(* CoDeSys 2.3.9.35 project: Controle de Nível com sensor analógico e IHM.pro *)
(* Author: Altus *)
(* Libraries: DU35x.lib 7.7.11 15:59:13, Navigation.lib 15.7.11 10:06:00, SysLibTargetVisu.lib 26.11.08 09:53:28, Standard.lib 26.11.08 09:46:20, Iecsfc.lib 26.11.08 09:46:14, SYSLIBCALLBACK.LIB 26.11.08 09:53:30 *)

(* PLC configuration (modules and I/O channels)
Comunicação [Comunica] node 0, in %IB0 out %QB0
  COM1 [COM1] node 0, in %IB0 out %QB0 {BaudRate = 115200; Paridade = Sem Paridade; StopBits = 1 Stop Bit; Modem = Sem RTS/CTS; Delay = 5}
    MToolIEC [Codesys] node 0, in %IB0 out %QB0
  COM2 [COM2] node 1, in %IB0 out %QB0 {BaudRate = 115200; Paridade = Sem Paridade; StopBits = 1 Stop Bit; Modem = Sem RTS/CTS; Delay = 5}
    Desabilitada [Desabilitado485] node 0, in %IB0 out %QB0
Entradas Digitais 0 [Entradas0] node 0, in %IW0 out %QB0
  I00 AT %IX0.0 [BitInput] I0.0
  I01 AT %IX0.1 [BitInput] I0.1
  I02 AT %IX0.2 [BitInput] I0.2
  I03 AT %IX0.3 [BitInput] I0.3
  I04 AT %IX0.4 [BitInput] I0.4
  I05 AT %IX0.5 [BitInput] I0.5
  I06 AT %IX0.6 [BitInput] I0.6
  I07 AT %IX0.7 [BitInput] I0.7
  I08 AT %IX0.8 [BitInput] I0.8
Entradas Digitais 1 [Entradas1] node 0, in %IW1 out %QB0
  I10 AT %IX1.0 [BitInput] I1.0
  I11 AT %IX1.1 [BitInput] I1.1
  I12 AT %IX1.2 [BitInput] I1.2
  I13 AT %IX1.3 [BitInput] I1.3
  I14 AT %IX1.4 [BitInput] I1.4
  I15 AT %IX1.5 [BitInput] I1.5
  I16 AT %IX1.6 [BitInput] I1.6
  I17 AT %IX1.7 [BitInput] I1.7
  I18 AT %IX1.8 [BitInput] I1.8
Entradas Digitais 2 [Entradas2] node 0, in %IW2 out %QB0
  I20 AT %IX2.0 [BitInput] I2.0
  I21 AT %IX2.1 [BitInput] I2.1
AI0 AT %IW4 [WordInput] AI0 {TipoAnalogica = Tensão 0-10V; FiltroAnalogica = Filtro 0 - AI=2ms  / AV=90ms; FundoEscala = 100}
AI1 AT %IW5 [WordInput] AI1 {TipoAnalogica = Channel Disable; FiltroAnalogica = Filter 0 - AI=2ms  / AV=90ms; FundoEscala = 0}
AI2 AT %IW6 [WordInput] AI2 {TipoAnalogica = Channel Disable; FiltroAnalogica = Filter 0 - AI=2ms  / AV=90ms; FundoEscala = 0}
AI3 AT %IW7 [WordInput] AI3 {TipoAnalogica = Channel Disable; FiltroAnalogica = Filter 0 - AI=2ms  / AV=90ms; FundoEscala = 0}
Entradas Rápidas [EntradasRapidas] node 1, in %IB16 out %QB0
  Bloco 0 [Bloco0] node 0, in %IB16 out %QB0
    Desabilitado [DesabilitadoBloco0] node 0, in %IB16 out %QB0
  Bloco 1 [Bloco1] node 1, in %IB16 out %QB0
    Desabilitado [DesabilitadoBloco1] node 0, in %IB16 out %QB0
  Entrada Configuravél Bloco 0 [EntradaConfiBloco0] node 2, in %IB16 out %QB0
    Contador 0 [EntradaConfContador0] node 0, in %IB16 out %QB0 {EntradaConfiguravelContador = Disable}
  Entrada Configuravél Bloco 1 [EntradaConfiBloco1] node 3, in %IB16 out %QB0
    Contador 2 [EntradaConfContador2] node 0, in %IB16 out %QB0 {EntradaConfiguravelContador = Disable}
Saídas [Saidas] node 1, in %IB13 out %QB0
  Saídas Digitais 0 [Saidas0] node 0, in %IW0 out %QW0
    Q00 AT %QX0.0 [BitOutput] Q0.0
    Q01 AT %QX0.1 [BitOutput] Q0.1
    Q02 AT %QX0.2 [BitOutput] Q0.2
    Q03 AT %QX0.3 [BitOutput] Q0.3
    Q04 AT %QX0.4 [BitOutput] Q0.4
    Q05 AT %QX0.5 [BitOutput] Q0.5
    Q06 AT %QX0.6 [BitOutput] Q0.6
    Q07 AT %QX0.7 [BitOutput] Q0.7
  Saídas Digitais 1 [Saidas1] node 0, in %IW0 out %QW1
    Q10 AT %QX1.0 [BitOutput] Q1.0
    Q11 AT %QX1.1 [BitOutput] Q1.1
    Q12 AT %QX1.2 [BitOutput] Q1.2
    Q13 AT %QX1.3 [BitOutput] Q1.3
    Q14 AT %QX1.4 [BitOutput] Q1.4
    Q15 AT %QX1.5 [BitOutput] Q1.5
    Q16 AT %QX1.6 [BitOutput] Q1.6
    Q17 AT %QX1.7 [BitOutput] Q1.7
  Saídas Analógicas [SaidaAnalogica] node 0, in %IW0 out %QW3
    AO0 AT %QW3 [WordOutput] AO0 {TipoAnalogica = Channel Disable; FundoEscala = 0}
    AO1 AT %QW4 [WordOutput] AO1 {TipoAnalogica = Channel Disable; FundoEscala = 0}
  Saídas Rápidas [SaidasRapidas] node 1, in %IB0 out %QB10
    Saída Rápida 0 Desabilitada [DesabilitadoF0] node 0, in %IB0 out %QB10
    Saída Rápida 1 Desabilitada [DesabilitadoF1] node 1, in %IB0 out %QB10
  Saídas Comum de Contador [SaidasContador] node 2, in %IB0 out %QB10
    Saída do Bloco 0 Desabilitada [DesabilitadoSaidaBloco0] node 0, in %IB0 out %QB10
    Saída do Bloco 1 Desabilitada [DesabilitadoSaidaBloco1] node 1, in %IB0 out %QB10
Eventos Externos [Eventos] node 2, in %IB13 out %QB6
  Evento Temporizado [TimerEvent] node 0, in %IB13 out %QB6 {Intervalo = 10}
*)

(* Task configuration *)
TASK PRINCIPAL (PRIORITY := 1, INTERVAL := T#1ms);
	PLC_PRG();
END_TASK
TASK NAVIGATION (PRIORITY := 1, INTERVAL := T#20ms);
	NAVEGA();
END_TASK
TASK VISUALIZATION (PRIORITY := 1, INTERVAL := T#500ms);
	MAINTARGETVISU_PAINT_CODE
END_TASK
TASK KEYBOARD_USAGE (PRIORITY := 1, INTERVAL := T#20ms);
	MAINTARGETVISU_INPUT_CODE
END_TASK

(* POU PLC_PRG, LD *)
PROGRAM PLC_PRG
VAR
	Desliga AT %IX0.0: BOOL; (* Botão B0 - NF: Desliga o controle de nível *)
	Liga AT %IX0.1: BOOL; (* Botão B1 - NA: Liga o controle de nível *)
	RT1 AT %IX0.2: BOOL;  (* Relé térmico RT1 - NF *)
	RT2 AT %IX0.3: BOOL;  (* Relé térmico RT2 - NF *)

	LG AT %QX1.0: BOOL; (* Lâmpada verde: Bomba desligada *)
	LY AT %QX1.1: BOOL; (* Lâmpada amarela: Térmico atuado ou nível alto *)
	LR AT %QX1.2: BOOL; (* Lâmpada vermelha: Bomba ligada em baixa ou alta rotação *)

	K1 AT %QX1.3: BOOL; (* Contator K1: Liga o motor em baixa rotação *)
	K2 AT %QX1.4: BOOL; (* Contator K2: Liga o motor em alta rotação *)
	K3 AT %QX1.5: BOOL; (* Contator K3: Liga o motor em alta rotação *)

	NivelBaixo: INT := 50; 	 (* Variável para armazenar o valor do nível baixo em litros *)
	NivelAlto: INT := 90; 	 (* Variável para armazenar o valor do nível alto em litros *)
	Overflow: BOOL := FALSE; (* Variável para armazenar o estado de transbordamento do tanque *)

	(* Variável para armazenar o nivel de rotação da bomba *)
	Slow : BOOL := FALSE;	(* Variável para armazenar o estado de baixa rotação do motor *)
	Fast : BOOL := FALSE;	(* Variável para armazenar o estado de alta rotação do motor *)
	Hot: BOOL := FALSE; 	(* Variável para armazenar o estado de superaquecimento do motor *)

	T : TIME := T#500ms; (* Tempo para piscar as lâmpadas *)
	TLY1 : TON; (* Temporizador para piscar a lâmpada amarela *)
	TLY2 : TON;
	TLR1 : TON; (* Temporizador para piscar a lâmpada vermelha *)
	TLR2 : TON;

	Estado : BOOL; 		(* Variável para armazenar o estado do sistema *)
	Emergencia : BOOL;  (* Variável para armazenar o estado de emergência *)
END_VAR
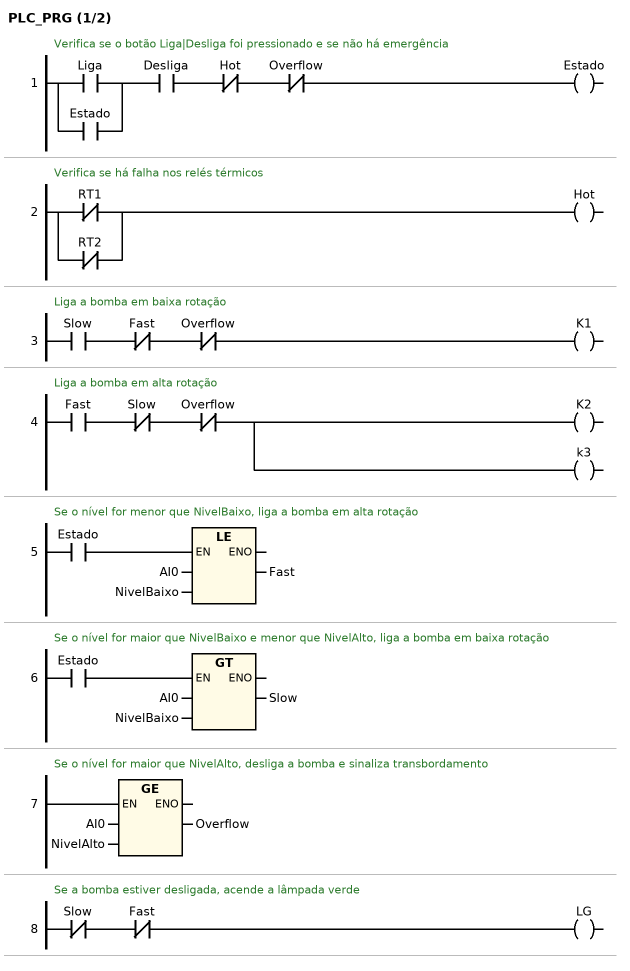
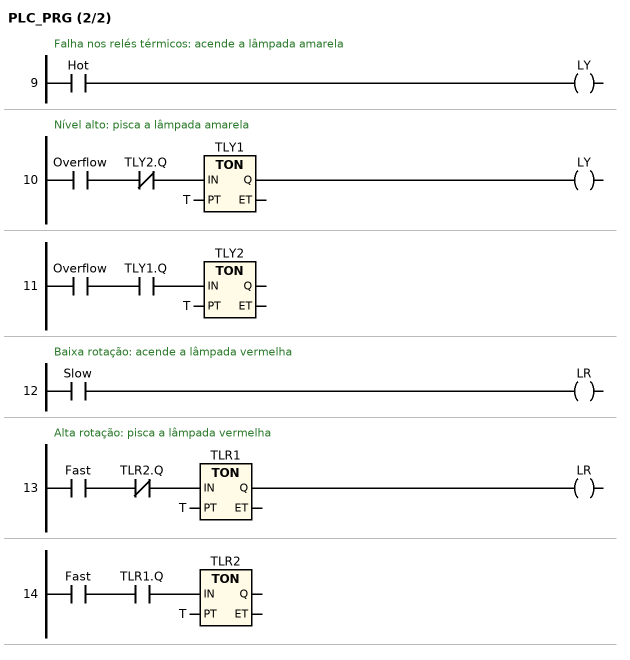
_LD_ (* Ladder Diagram *)
NETWORK 1 (* Verifica se o botão Liga|Desliga foi pressionado e se não há emergência *)
	{ [Liga] | [Estado] } - [Desliga] - [/Hot] - [/Overflow] --- (Estado)
NETWORK 2 (* Verifica se há falha nos relés térmicos *)
	{ [/RT1] | [/RT2] } --- (Hot)
NETWORK 3 (* Liga a bomba em baixa rotação *)
	[Slow] - [/Fast] - [/Overflow] --- (K1)
NETWORK 4 (* Liga a bomba em alta rotação *)
	[Fast] - [/Slow] - [/Overflow] --- (K2) (k3)
NETWORK 5 (* Se o nível for menor que NivelBaixo, liga a bomba em alta rotação *)
	[Estado]
		EN --- LE(AI0, NivelBaixo) => Fast
NETWORK 6 (* Se o nível for maior que NivelBaixo e menor que NivelAlto, liga a bomba em baixa rotação *)
	[Estado]
		EN --- GT(AI0, NivelBaixo) => Slow
NETWORK 7 (* Se o nível for maior que NivelAlto, desliga a bomba e sinaliza transbordamento *)
	*
		EN --- GE(AI0, NivelAlto) => Overflow
NETWORK 8 (* Se a bomba estiver desligada, acende a lâmpada verde *)
	[/Slow] - [/Fast] --- (LG)
NETWORK 9 (* Falha nos relés térmicos: acende a lâmpada amarela *)
	[Hot] --- (LY)
NETWORK 10 (* Nível alto: pisca a lâmpada amarela *)
	[Overflow] - [/TLY2.Q] - TLY1:TON(IN: *, PT: T) --- (LY)
NETWORK 11
	[Overflow] - [TLY1.Q] - TLY2:TON(IN: *, PT: T)
NETWORK 12 (* Baixa rotação: acende a lâmpada vermelha *)
	[Slow] --- (LR)
NETWORK 13 (* Alta rotação: pisca a lâmpada vermelha *)
	[Fast] - [/TLR2.Q] - TLR1:TON(IN: *, PT: T) --- (LR)
NETWORK 14
	[Fast] - [TLR1.Q] - TLR2:TON(IN: *, PT: T)
_END_LD_
(* the same logic as Structured Text *)
(* Network 1: Verifica se o botão Liga|Desliga foi pressionado e se não há emergência *)
Estado := (Liga OR Estado) AND Desliga AND NOT Hot AND NOT Overflow;
(* Network 2: Verifica se há falha nos relés térmicos *)
Hot := NOT RT1 OR NOT RT2;
(* Network 3: Liga a bomba em baixa rotação *)
K1 := Slow AND NOT Fast AND NOT Overflow;
(* Network 4: Liga a bomba em alta rotação *)
K2 := Fast AND NOT Slow AND NOT Overflow;
k3 := K2;
(* Network 5: Se o nível for menor que NivelBaixo, liga a bomba em alta rotação *)
IF Estado THEN
	Fast := AI0 <= NivelBaixo;
END_IF;
(* Network 6: Se o nível for maior que NivelBaixo e menor que NivelAlto, liga a bomba em baixa rotação *)
IF Estado THEN
	Slow := AI0 > NivelBaixo;
END_IF;
(* Network 7: Se o nível for maior que NivelAlto, desliga a bomba e sinaliza transbordamento *)
Overflow := AI0 >= NivelAlto;
(* Network 8: Se a bomba estiver desligada, acende a lâmpada verde *)
LG := NOT Slow AND NOT Fast;
(* Network 9: Falha nos relés térmicos: acende a lâmpada amarela *)
LY := Hot;
(* Network 10: Nível alto: pisca a lâmpada amarela *)
TLY1(IN := Overflow AND NOT TLY2.Q, PT := T);
LY := TLY1.Q;
(* Network 11 *)
TLY2(IN := Overflow AND TLY1.Q, PT := T);
(* Network 12: Baixa rotação: acende a lâmpada vermelha *)
LR := Slow;
(* Network 13: Alta rotação: pisca a lâmpada vermelha *)
TLR1(IN := Fast AND NOT TLR2.Q, PT := T);
LR := TLR1.Q;
(* Network 14 *)
TLR2(IN := Fast AND TLR1.Q, PT := T);
END_PROGRAM

(* POU NAVEGA, ST *)
PROGRAM NAVEGA
VAR
	ControleTelas : NAVIGATION;
	ListaTelas 	: ARRAY [0..30] OF STRING(10);
END_VAR
(* Adiciona a tela MAIN como tela principal *)
ListaTelas[0] := 'MAIN';

(* Ativa o controle automático de navegação somente pelo teclado *)
ControleTelas(ENABLE_UPDW := FALSE, VISU_LIST := ListaTelas, UP := FALSE , DOWN := FALSE);
END_PROGRAM
